FUNCTION_BLOCK el7xxxBasicAxis_FB EXTENDS BeckHoffBasicAxis_FB
VAR_INPUT
	pDigIn: 	POINTER TO INT;	
END_VAR
VAR_OUTPUT
END_VAR
VAR
	
END_VAR


AxisCtrlPtr^.Input.Parameter.Drive.eDriveType := enumDriveType.eEL70xx;
AxisCtrlPtr^.Input.Parameter.Drive.VendorNameID := eVendorNameID.Beckhoff;


SUPER^(AxisRef:=AxisRef);

IF (pDigIn <> 0) THEN
	AxisCtrlPtr^.Output.Status.DriveEnable	:= pDigIn^.7;
ELSE
	AxisCtrlPtr^.Output.Status.DriveEnable	:= TRUE;
END_IF

METHOD HomeLagErrExternFeedBack : BOOL
VAR_INPUT
	Execute: BOOL;
END_VAR

VAR_INST
	fbEcCoeSdoWriteMaxCurrent	: FB_EcCoeSdoWrite;
	State:INT;	
	ExtLagErrPrevState : INT;
	HomeTrig: Trigger;
	Reset:BOOL;	
	Delay:	TON;	
	LastActExternEncodPos:		UDINT;
	DiffExternEncodPos:			DINT;
	LatchSetPos:				LREAL;			
	CalckedLagError:			LREAL;
	EncdSampleTimer:			TON;
	StartPosMonitor:			BOOL;
		
END_VAR
Reset:= Execute;
IF HomeTrig.EDGEPOS(Reset) THEN
	Reset:=	FALSE;
	State:=1;
	
	HomeLagErrExternFeedBack:= FALSE ;
	HomingActive:= 	TRUE ;
	AxisCtrlPtr^.Output.Status.MC_Home.Done:= FALSE ;
	fbMC_MoveVel.Execute:= FALSE ;
	fbMC_MoveRel.Execute:= FALSE ;
END_IF

IF Execute THEN
	CASE State OF
		
		1:									
			fbEcCoeSdoWriteMaxCurrent.sNetId:= 		strEcNetId;
			fbEcCoeSdoWriteMaxCurrent.nSlaveAddr:= 	AxisCtrlPtr^.Input.Parameter.Drive.EtherCatAddr;
			fbEcCoeSdoWriteMaxCurrent.nSubIndex:=	1;
			fbEcCoeSdoWriteMaxCurrent.nIndex:= 		16#8010;  			
			fbEcCoeSdoWriteMaxCurrent.pSrcBuf:=		 ADR(AxisCtrlPtr^.Input.Parameter.HomeOptions.stLagErr.BlockSearchMaxCurrent); 
			fbEcCoeSdoWriteMaxCurrent.cbBufLen:= 	SIZEOF(AxisCtrlPtr^.Input.Parameter.HomeOptions.stLagErr.BlockSearchMaxCurrent); 
			fbEcCoeSdoWriteMaxCurrent.bExecute:= 	TRUE; 
			fbEcCoeSdoWriteMaxCurrent.tTimeout:= 	T#2S;					
			State:= State +1;							
			 
		2:		
			IF NOT fbEcCoeSdoWriteMaxCurrent.bBusy THEN
				fbEcCoeSdoWriteMaxCurrent.bExecute:= FALSE;
				IF NOT fbEcCoeSdoWriteMaxCurrent.bError THEN																									
					State:= State +1;
				ELSE
					fbEcCoeSdoWriteMaxCurrent.bExecute:= FALSE;
					fnLogMsg(ADR(LogMsg_0),LOG_ERROR,Concat('ADS Error Code %d: ',F_ADStoStr(fbEcCoeSdoWriteMaxCurrent.nErrId)),UDINT_TO_DINT(fbEcCoeSdoWriteMaxCurrent.nErrId),0,0);
					State:= 0;				
				END_IF				
			END_IF 		 
		3:	
			IF WriteNC_AxisBoolParam(MC_AxisParameter:=MC_AxisParameter.EnablePosLagMonitoring,ParamValue:=FALSE) THEN
				State:= State +1;	
			END_IF
						
										
		4: 										
			IF AxisCtrlPtr^.Input.Parameter.HomeOptions.stBasic.StartDirection = eHomeModeOption.eNEGATIVE THEN								
				fbMC_MoveVel.Direction:= 	MC_Negative_Direction; 					
			ELSIF AxisCtrlPtr^.Input.Parameter.HomeOptions.stBasic.StartDirection = eHomeModeOption.ePOSITIVE THEN								
				fbMC_MoveVel.Direction:= 	MC_Positive_Direction;										
			END_IF
			
			fbMC_MoveVel.Velocity:= AxisCtrlPtr^.Input.Parameter.HomeOptions.stBasic.SwitchVelo;			
			fbMC_MoveVel.Execute:= 	TRUE ;
			LastActExternEncodPos:=	AxisCtrlPtr^.Output.monitor.ActExternEncodPos;						
			State:= State + 1;
			
		5:	IF AxisCtrlPtr^.Output.Status.AxisStatus.ContinuousMotion THEN
				EncdSampleTimer(IN:= NOT(EncdSampleTimer.Q),PT:=T#0.2S);
				IF EncdSampleTimer.Q THEN	
					State:= State + 1;
				END_IF	
			END_IF
		6: 							
			DiffExternEncodPos:=ABS(UDINT_TO_DINT(AxisCtrlPtr^.Output.monitor.ActExternEncodPos) - UDINT_TO_DINT(LastActExternEncodPos));
			IF DiffExternEncodPos <= 4 THEN
				LatchSetPos:=	AxisCtrlPtr^.Output.monitor.ActPosition;			
				State:= State + 1;
			ELSE
				LastActExternEncodPos:=	AxisCtrlPtr^.Output.monitor.ActExternEncodPos;	
				State:= 5;
			END_IF			
					
		7:									
			CalckedLagError:=	ABS(AxisCtrlPtr^.Output.monitor.ActPosition - LatchSetPos);										
			IF (CalckedLagError > AxisCtrlPtr^.Input.Parameter.HomeOptions.stLagErr.LagErr) THEN
				State:= State + 1;	
			END_IF
			
		
		8:	
			IF Stop() THEN
				State:= State + 1;				
			END_IF
					
		9:	InternalPowerHandle:=	TRUE;
			AxisCtrlPtr^.Input.Command.Power:= FALSE;
			IF AxisCtrlPtr^.Output.Status.AxisStatus.Disabled THEN
				State:= State + 1;	
			END_IF
			
		10:	Delay(IN:=	TRUE,PT:=T#0.5S);		
			IF Delay.Q THEN
				Delay(IN:=FALSE);	
				State:= State +1;
			END_IF
			
		11:	InternalPowerHandle:=	FALSE;
			AxisCtrlPtr^.Input.Command.Power:= TRUE;
			State:= State +1;
		
		12:	
	
			IF (AxisCtrlPtr^.Output.Status.MC_Power.Status = TRUE) THEN
				State:= State + 1;	
			END_IF
			
			
		13:	Delay(IN:=	TRUE,PT:=T#0.5S);		
			IF Delay.Q THEN
				Delay(IN:=FALSE);
					
				State:= State +1;
			END_IF
			
		14:		
		

			IF fbEcCoeSdoWriteMaxCurrent.bBusy = FALSE THEN
				fbEcCoeSdoWriteMaxCurrent.sNetId:= 		strEcNetId;
				fbEcCoeSdoWriteMaxCurrent.nSlaveAddr:= 	AxisCtrlPtr^.Input.Parameter.Drive.EtherCatAddr;
				fbEcCoeSdoWriteMaxCurrent.nSubIndex:=	1;
				fbEcCoeSdoWriteMaxCurrent.nIndex:= 		16#8010;  				
				fbEcCoeSdoWriteMaxCurrent.pSrcBuf:=		 ADR(AxisCtrlPtr^.Input.Parameter.HomeOptions.stLagErr.BlockExitMaxCurrent); 				
				fbEcCoeSdoWriteMaxCurrent.cbBufLen:= 	SIZEOF(AxisCtrlPtr^.Input.Parameter.HomeOptions.stLagErr.BlockExitMaxCurrent); 
				fbEcCoeSdoWriteMaxCurrent.bExecute:= 	TRUE; 
				fbEcCoeSdoWriteMaxCurrent.tTimeout:= 	T#2S;	
								
				
				State:= State +1;				
			END_IF
			
			
			
							
		15:		
			State:= State +1;
		16:	
			IF NOT fbEcCoeSdoWriteMaxCurrent.bBusy THEN
				fbEcCoeSdoWriteMaxCurrent.bExecute:= FALSE;
				IF NOT fbEcCoeSdoWriteMaxCurrent.bError THEN																									
					State:= State +1;
				ELSE
					fbEcCoeSdoWriteMaxCurrent.bExecute:= FALSE;
					fnLogMsg(ADR(LogMsg_0),LOG_ERROR,Concat('ADS Error Code %d: ',F_ADStoStr(fbEcCoeSdoWriteMaxCurrent.nErrId)),UDINT_TO_DINT(fbEcCoeSdoWriteMaxCurrent.nErrId),0,0);
					State:= 0;				
				END_IF				
			END_IF 		 
				
		17:	
			IF WriteNC_AxisBoolParam(MC_AxisParameter:=MC_AxisParameter.EnablePosLagMonitoring,ParamValue:=FALSE) THEN			
				State:= State +1;	
			END_IF	
			
														
		18:		
			fbMC_Home.HomingMode:= 	MC_Direct ;
			fbMC_Home.Position:= 	0;
			fbMC_Home.Execute:= 	TRUE;	
			State:= State + 1;
							
		19:	
			IF fbMC_Home.Done THEN
				fbMC_Home.Execute := FALSE;		
				IF AxisCtrlPtr^.Input.Parameter.HomeOptions.stBasic.StartDirection = eHomeModeOption.eNEGATIVE THEN													
					fbMC_MoveRel.Distance:=		AxisCtrlPtr^.Input.Parameter.HomeOptions.stLagErr.TriggerOffsetPos ;					
				ELSIF AxisCtrlPtr^.Input.Parameter.HomeOptions.stBasic.StartDirection = eHomeModeOption.ePOSITIVE THEN								
					fbMC_MoveRel.Distance:=		AxisCtrlPtr^.Input.Parameter.HomeOptions.stLagErr.TriggerOffsetPos*(-1) ;											
				END_IF
				fbMC_MoveRel.Velocity:= AxisCtrlPtr^.Input.Parameter.HomeOptions.stBasic.TriggerVelo;
				
				fbMC_MoveRel.Execute:= 	TRUE ;
				State:= State + 1;	
			END_IF
			
		20:	IF fbMC_MoveRel.Done THEN
				fbMC_MoveRel.Execute := FALSE;
				fbMC_Home.HomingMode:= 	MC_Direct ;
				//fbMC_Home.Options:= 	AxisCtrlPtr^.Input.Parameter.HomeOptions.NcHomeOption;
				fbMC_Home.Position:= 	(AxisCtrlPtr^.Input.Parameter.HomeOptions.stBasic.HomeSetPos) * (-1); 
				fbMC_Home.Execute:= 	TRUE;	
				State := 100 ;
			END_IF
																											
		100:
			IF fbMC_Home.Done THEN
				AxisCtrlPtr^.Input.Command.Home:= FALSE ;
				HomingActive:= 							FALSE;
				HomeLagErrExternFeedBack:= 		TRUE;
				fbMC_Home.Execute:= 					FALSE;
				AxisCtrlPtr^.Output.Status.MC_Home.Done:= TRUE ;
				State:= 0;
			END_IF
	END_CASE
	IF ExtLagErrPrevState <> State THEN
		fnLogMsg(ADR(LogMsg_0),LOG_INFO,'Drive Lag Err step %d',State,0,0);
		ExtLagErrPrevState := State;
	END_IF	
	
END_IF
 

fbMC_MoveVel.Acceleration  	:= AxisCtrlPtr^.Input.Parameter.Acceleration;
fbMC_MoveVel.Deceleration  	:= AxisCtrlPtr^.Input.Parameter.Deceleration;
fbMC_MoveVel.Jerk			:= AxisCtrlPtr^.Input.Parameter.Jerk;
fbMC_MoveVel.Options		:= AxisCtrlPtr^.Input.Parameter.Options;
fbMC_MoveVel.BufferMode		:= AxisCtrlPtr^.Input.Parameter.BufferMode;

fbMC_MoveRel.Acceleration  	:= AxisCtrlPtr^.Input.Parameter.Acceleration;
fbMC_MoveRel.Deceleration  	:= AxisCtrlPtr^.Input.Parameter.Deceleration;
fbMC_MoveRel.Jerk			:= AxisCtrlPtr^.Input.Parameter.Jerk;
fbMC_MoveRel.Options		:= AxisCtrlPtr^.Input.Parameter.Options;
fbMC_MoveRel.BufferMode		:= AxisCtrlPtr^.Input.Parameter.BufferMode;

{warning disable C0371}
//Warning: Access to VAR_IN_OUT <Var> declared in <POU> from external context <Method/Transition/Property>
fbMC_Home(Axis:= AxisRef);	
fbMC_MoveVel(Axis:= AxisRef);
fbMC_MoveRel(Axis:= AxisRef);


fbMC_Stop.Deceleration:= 	AxisCtrlPtr^.Input.Parameter.Deceleration;
fbMC_Stop.Jerk:=			AxisCtrlPtr^.Input.Parameter.Jerk;
fbMC_Stop.Options:= 		AxisCtrlPtr^.Input.Parameter.Options;
fbMC_Stop(Axis := AxisRef) ;
{warning restore C0371}

fbEcCoeSdoWriteMaxCurrent();

THIS^.HomingGlobalHandle();
END_METHOD

METHOD HomeLagErrInternalEnc : BOOL
VAR_INPUT
	Execute: BOOL;
END_VAR

VAR_INST
	fbEcCoeSdoWriteMaxCurrent	: FB_EcCoeSdoWrite;
//	State:INT;	
//	HomeTrig: Trigger;
//	Reset:BOOL;	
//	Delay:	TON;	
END_VAR
Reset:= Execute;
IF HomeTrig.EDGEPOS(Reset) THEN
	Reset:=	FALSE;
	State:=1;
	HomeLagErrInternalEnc:= FALSE ;
	HomingActive:= 	TRUE ;
	AxisCtrlPtr^.Output.Status.MC_Home.Done:= FALSE ;
	fbMC_MoveVel.Execute:= FALSE ;
	fbMC_MoveRel.Execute:= FALSE ;
END_IF

IF Execute THEN
	CASE State OF
		
		1:									
			fbEcCoeSdoWriteMaxCurrent.sNetId:= 		strEcNetId;
			fbEcCoeSdoWriteMaxCurrent.nSlaveAddr:= 	AxisCtrlPtr^.Input.Parameter.Drive.EtherCatAddr;
			fbEcCoeSdoWriteMaxCurrent.nSubIndex:=	1;
			fbEcCoeSdoWriteMaxCurrent.nIndex:= 		16#8010;  
			fbEcCoeSdoWriteMaxCurrent.pSrcBuf:=		 ADR(AxisCtrlPtr^.Input.Parameter.HomeOptions.stLagErr.BlockSearchMaxCurrent); 
			fbEcCoeSdoWriteMaxCurrent.cbBufLen:= 	SIZEOF(AxisCtrlPtr^.Input.Parameter.HomeOptions.stLagErr.BlockSearchMaxCurrent); 
			fbEcCoeSdoWriteMaxCurrent.bExecute:= 	TRUE; 
			fbEcCoeSdoWriteMaxCurrent.tTimeout:= 	T#2S;					
			State:= State +1;
				
			//IF (NOT SDOrw.Output.Status.EcCoeSdoWrite.bError) THEN
			//	SDOrw.Input.Command.EcCoeSdoWrite.Enable:= TRUE;
			//END_IF
			//SDOrw.Input.Parameter.EcCoeSdoWrite.sNetId 		:= strEcNetId;
		    //SDOrw.Input.Parameter.EcCoeSdoWrite.nSlaveAddr	:= AxisCtrlPtr^.Input.Parameter.nSlaveAddr;
			//SDOrw.Input.Parameter.EcCoeSdoWrite.nIndex		:= 	16#8010;	
		    //SDOrw.Input.Parameter.EcCoeSdoWrite.nSubIndex	:= 	1; 			
			//SDOrw.Input.Parameter.EcCoeSdoWrite.pSrcBuf		:=  ADR(AxisCtrlPtr^.Input.Parameter.HomeOptions.BlockSearchMaxCurrent); 
			//SDOrw.Input.Parameter.EcCoeSdoWrite.cbBufLen	:=  SIZEOF(AxisCtrlPtr^.Input.Parameter.HomeOptions.BlockSearchMaxCurrent);		
			//State:= State +1;
			 
		2:
			//IF THIS^.EcCoeSdoWrite() THEN 
			//	 State:= State +1;
			// END_IF	
			IF NOT fbEcCoeSdoWriteMaxCurrent.bBusy THEN
				fbEcCoeSdoWriteMaxCurrent.bExecute:= FALSE;
				IF NOT fbEcCoeSdoWriteMaxCurrent.bError THEN																									
					State:= State +1;
				ELSE
					fbEcCoeSdoWriteMaxCurrent.bExecute:= FALSE;
					fnLogMsg(ADR(LogMsg_0),LOG_ERROR,Concat('int ADS Error Code %d index-0x8010: ',F_ADStoStr(fbEcCoeSdoWriteMaxCurrent.nErrId)),UDINT_TO_DINT(fbEcCoeSdoWriteMaxCurrent.nErrId),0,0);
					State:= 0;				
				END_IF				
			END_IF 		 
		3:	
			IF WriteNC_AxisBoolParam(MC_AxisParameter:=MC_AxisParameter.EnablePosLagMonitoring,ParamValue:=FALSE) THEN
				State:= State +1;	
			END_IF
						
										
		4: 										
			IF AxisCtrlPtr^.Input.Parameter.HomeOptions.stBasic.StartDirection = eHomeModeOption.eNEGATIVE THEN								
				fbMC_MoveVel.Direction:= 	MC_Negative_Direction; 					
			ELSIF AxisCtrlPtr^.Input.Parameter.HomeOptions.stBasic.StartDirection = eHomeModeOption.ePOSITIVE THEN								
				fbMC_MoveVel.Direction:= 	MC_Positive_Direction;										
			END_IF
			
			fbMC_MoveVel.Velocity:= AxisCtrlPtr^.Input.Parameter.HomeOptions.stBasic.SwitchVelo;
	
			fbMC_MoveVel.Execute:= 	TRUE ;
			
			State:= State + 1;
			
		5: 	
			IF (ABS(AxisCtrlPtr^.Output.monitor.ActLagError) > AxisCtrlPtr^.Input.Parameter.HomeOptions.stLagErr.LagErr) THEN
				State:= State + 1;	
			END_IF
		
		6:	
			IF Stop() THEN
				State:= State + 1;				
			END_IF
					
		7:	InternalPowerHandle:=	TRUE;
			AxisCtrlPtr^.Input.Command.Power:= FALSE;
			IF AxisCtrlPtr^.Output.Status.AxisStatus.Disabled THEN
				State:= State + 1;	
			END_IF
			
		8:	Delay(IN:=	TRUE,PT:=T#1S);		
			IF Delay.Q THEN
				Delay(IN:=FALSE);	
				State:= State +1;
			END_IF
			
		9:	InternalPowerHandle:=	FALSE;
			AxisCtrlPtr^.Input.Command.Power:= TRUE;
			IF (AxisCtrlPtr^.Output.Status.AxisStatus.Disabled = FALSE) THEN
				State:= State + 1;	
			END_IF
			
			
		10:	
		(*
			IF (NOT SDOrw.Output.Status.EcCoeSdoWrite.bError) THEN
				SDOrw.Input.Command.EcCoeSdoWrite.Enable 		:= TRUE;
			END_IF
			SDOrw.Input.Parameter.EcCoeSdoWrite.sNetId 		:= strEcNetId;
		    SDOrw.Input.Parameter.EcCoeSdoWrite.nSlaveAddr	:= LREAL_TO_UINT(AxisCtrlPtr^.Input.Parameter.Drive.EtherCatAddr.Value);
			SDOrw.Input.Parameter.EcCoeSdoWrite.nIndex		:= 	16#8010;	
		    SDOrw.Input.Parameter.EcCoeSdoWrite.nSubIndex	:= 	1; 			
			SDOrw.Input.Parameter.EcCoeSdoWrite.pSrcBuf		:=  ADR(AxisCtrlPtr^.Input.Parameter.HomeOptions.stLagErr.BlockExitMaxCurrent); 
			SDOrw.Input.Parameter.EcCoeSdoWrite.cbBufLen	:=  SIZEOF(AxisCtrlPtr^.Input.Parameter.HomeOptions.stLagErr.BlockExitMaxCurrent);	
		*)
			
			fbEcCoeSdoWriteMaxCurrent.sNetId:= 		strEcNetId;
			fbEcCoeSdoWriteMaxCurrent.nSlaveAddr:= AxisCtrlPtr^.Input.Parameter.Drive.EtherCatAddr;
			fbEcCoeSdoWriteMaxCurrent.nSubIndex:= 1;
			fbEcCoeSdoWriteMaxCurrent.nIndex:= 		16#8010;
			fbEcCoeSdoWriteMaxCurrent.pSrcBuf:=		ADR(AxisCtrlPtr^.Input.Parameter.HomeOptions.stLagErr.BlockExitMaxCurrent); 
			fbEcCoeSdoWriteMaxCurrent.cbBufLen:= SIZEOF(AxisCtrlPtr^.Input.Parameter.HomeOptions.stLagErr.BlockExitMaxCurrent);
			fbEcCoeSdoWriteMaxCurrent.bExecute:=  TRUE;
			fbEcCoeSdoWriteMaxCurrent.tTimeout:= T#2S;
			
			State:= State +1; 

		11:	
			IF NOT fbEcCoeSdoWriteMaxCurrent.bBusy THEN
				fbEcCoeSdoWriteMaxCurrent.bExecute:= FALSE;		
				 State:= State +1;
			END_IF		
				
		12:	
			IF WriteNC_AxisBoolParam(MC_AxisParameter:=MC_AxisParameter.EnablePosLagMonitoring,ParamValue:=TRUE) THEN			
				State:= State +1;	
			END_IF	
			
														
		13:		
			fbMC_Home.HomingMode:= 	MC_Direct ;
			//fbMC_Home.Options:= 	AxisCtrlPtr^.Input.Parameter.HomeOptions.NcHomeOption ;
			fbMC_Home.Position:= 	0;
			fbMC_Home.Execute:= 	TRUE;	
			State:= State + 1;
							
		14:	
			IF fbMC_Home.Done THEN
				fbMC_Home.Execute := FALSE;		
				IF AxisCtrlPtr^.Input.Parameter.HomeOptions.stBasic.StartDirection = eHomeModeOption.eNEGATIVE THEN													
					fbMC_MoveRel.Distance:=		AxisCtrlPtr^.Input.Parameter.HomeOptions.stLagErr.TriggerOffsetPos ;					
				ELSIF AxisCtrlPtr^.Input.Parameter.HomeOptions.stBasic.StartDirection = eHomeModeOption.ePOSITIVE THEN								
					fbMC_MoveRel.Distance:=		AxisCtrlPtr^.Input.Parameter.HomeOptions.stLagErr.TriggerOffsetPos*(-1) ;											
				END_IF
				fbMC_MoveRel.Velocity:= AxisCtrlPtr^.Input.Parameter.HomeOptions.stBasic.TriggerVelo;
				
				fbMC_MoveRel.Execute:= 	TRUE ;
				State:= State + 1;	
			END_IF
			
		15:	IF fbMC_MoveRel.Done THEN
				fbMC_Home.HomingMode:= 	MC_Direct ;
				//fbMC_Home.Options:= 	AxisCtrlPtr^.Input.Parameter.HomeOptions.NcHomeOption;
				fbMC_Home.Position:= 	(AxisCtrlPtr^.Input.Parameter.HomeOptions.stBasic.HomeSetPos) * (-1); 
				fbMC_Home.Execute:= 	TRUE;	
				State := 100 ;
			END_IF
																											
		100:
			IF fbMC_Home.Done THEN
				AxisCtrlPtr^.Input.Command.Home:= FALSE ;
				HomingActive:= 				FALSE;
				HomeLagErrInternalEnc:= 		TRUE;
				fbMC_Home.Execute:= 		FALSE;
				AxisCtrlPtr^.Output.Status.MC_Home.Done:= TRUE ;
				State:= 0;
			END_IF
	END_CASE

END_IF
 

fbMC_MoveVel.Acceleration  	:= AxisCtrlPtr^.Input.Parameter.Acceleration;
fbMC_MoveVel.Deceleration  	:= AxisCtrlPtr^.Input.Parameter.Deceleration;
fbMC_MoveVel.Jerk			:= AxisCtrlPtr^.Input.Parameter.Jerk;
fbMC_MoveVel.Options		:= AxisCtrlPtr^.Input.Parameter.Options;
fbMC_MoveVel.BufferMode		:= AxisCtrlPtr^.Input.Parameter.BufferMode;

fbMC_MoveRel.Acceleration  	:= AxisCtrlPtr^.Input.Parameter.Acceleration;
fbMC_MoveRel.Deceleration  	:= AxisCtrlPtr^.Input.Parameter.Deceleration;
fbMC_MoveRel.Jerk			:= AxisCtrlPtr^.Input.Parameter.Jerk;
fbMC_MoveRel.Options		:= AxisCtrlPtr^.Input.Parameter.Options;
fbMC_MoveRel.BufferMode		:= AxisCtrlPtr^.Input.Parameter.BufferMode;

{warning disable C0371}
//Warning: Access to VAR_IN_OUT <Var> declared in <POU> from external context <Method/Transition/Property>

fbMC_Home(Axis:= AxisRef);	
fbMC_MoveVel(Axis:= AxisRef);
fbMC_MoveRel(Axis:= AxisRef);

fbMC_Stop.Deceleration:= 	AxisCtrlPtr^.Input.Parameter.Deceleration;
fbMC_Stop.Jerk:=			AxisCtrlPtr^.Input.Parameter.Jerk;
fbMC_Stop.Options:= 		AxisCtrlPtr^.Input.Parameter.Options;
fbMC_Stop(Axis := AxisRef) ;
{warning restore C0371}
fbEcCoeSdoWriteMaxCurrent();

THIS^.HomingGlobalHandle();
END_METHOD

METHOD HomeLagError : BOOL
VAR_INPUT
	Execute: BOOL;
END_VAR

VAR_INST
	LagErrorState : INT;
	HomingLagErrorTrig: Trigger;
END_VAR
VAR
	
END_VAR


IF HomingLagErrorTrig.EDGEPOS(Execute) THEN
	LagErrorState := 1;
	HomeLagError := FALSE;
END_IF


IF HomingLagErrorTrig.EDGENEG(Execute) THEN
	
	LagErrorState := 0;
	
END_IF

CASE LagErrorState OF
	 
	
	1:
		HomeLagErrExternFeedBack(FALSE);
		HomeLagErrInternalEnc(FALSE);
		LagErrorState := LagErrorState +1;
	2:
		IF AxisCtrlPtr^.Input.Parameter.HomeOptions.stBasic.ExternalEncoder THEN
			IF HomeLagErrExternFeedBack(TRUE) THEN
				LagErrorState := LagErrorState +1;				
			END_IF
		ELSE
			IF HomeLagErrInternalEnc(TRUE) THEN
				LagErrorState := LagErrorState +1;				
			END_IF
	
		END_IF		
	3:
		HomeLagError := TRUE;
	
END_CASE
END_METHOD

END_FUNCTION_BLOCK

(* stored: Version 1.1.0.1, ProductVersion 3.1.4024.3
   POU el7xxxBasicAxis_FB: Id {52d37af2-3990-0d87-268e-7fa97aeb215b}, SpecialFunc None
   Method HomeLagErrExternFeedBack: Id {824ad3ba-f315-00e8-3811-14e406adc2b4}
   Method HomeLagErrInternalEnc: Id {8bb3a084-d0f0-0f9a-366c-33d85a1e4478}
   Method HomeLagError: Id {588999a9-d6ce-0c30-23fa-0be6e6e13184} *)
